TYPE Motion_Parameters :
STRUCT
	
	
		maxAcceleration					: 		LREAL	:= 15000;			// mm/s^2
		
		maxVelocity						: 		LREAL	:= 50.0;			// mm/s
		
		minVelocity						: 		LREAL	:= -50.0;			// -mm/s
		
		RotationScailing				: 		LREAL 	:= 0.0002; 			// Radians/s^2
		
		deltaT							:		LREAL	:= 0.00025;			//Cycle time 

END_STRUCT
END_TYPE

(* stored: Version 1.1.0.1, ProductVersion 3.1.4024.12
   DUT Motion_Parameters: Id {8a77553b-194c-4510-ae1e-272b07e08d0a} *)
